// TIA Portal V21 export
TYPE "coneCrusherHMIs"
   STRUCT
      self { S7_SetPoint := 'True'} : "coneCrusherHMI";
      sg : "switchgearHMI";
      luS { S7_SetPoint := 'True'} : "lubricationSystemHMI";
   END_STRUCT;
END_TYPE
